{attribute addProperty BoxType "EL2642-0000-0016"}
{attribute addProperty Id "DO_Inputs_DeviceAT %I*DO_Inputs_Device_7B636AA11620DO_Group_1_OutputsAT %Q*DO_Group_1_Outputs_E2C7B95A1620DO_Group_2_OutputsAT %Q*DO_Group_2_Outputs_D5F4CCA31620WcStateAT %I*WcState_F855686C1620InfoDataAT %I*InfoData_0BDED7BF144180"}
{attribute addProperty CRC "2279681180"}
{attribute addProperty SizeInBites "208"}
{attribute addProperty SizeInBytes "26"}
TYPE EL2642_A8D73BA7 :
STRUCT
	{attribute addProperty Name "DO_Inputs_Device"}
	DO_Inputs_Device : DO_Inputs_Device_7B636AA1;
	{attribute addProperty Name "DO_Group_1_Outputs"}
	DO_Group_1_Outputs : DO_Group_1_Outputs_E2C7B95A;
	{attribute addProperty Name "DO_Group_2_Outputs"}
	DO_Group_2_Outputs : DO_Group_2_Outputs_D5F4CCA3;
	{attribute addProperty Name "WcState"}
	WcState : WcState_F855686C;
	{attribute addProperty Name "InfoData"}
	InfoData : InfoData_0BDED7BF;
END_STRUCT
END_TYPE

(* stored: Version 1.2.0.0, ProductVersion 3.1.4024.9
   DUT EL2642_A8D73BA7: Id {71e521b1-07ba-4564-ad0f-fa3e7994a6a6} *)
